TYPE ST_WorkTime :
STRUCT
	hours	: UDINT;
	minuts	: UINT;
	seconds	: UINT;
END_STRUCT
END_TYPE

(* stored: Version 1.1.0.1, ProductVersion 3.1.4024.12
   DUT ST_WorkTime: Id {775f549a-5109-4edc-b73b-2377fecf62db} *)
